// TIA Portal V20 export
DATA_BLOCK "LPFE_GlobalConfigurationData"   // DB240
TITLE = LPFE_GlobalConfigurationData
{ DB_Accessible_From_OPC_UA := 'FALSE' }
AUTHOR : DI FA SUP
FAMILY : LPFE
// Contains all global configurable settings
// stored: Access Published, DBAccessibleFromOPCUA false, DBAccessibleFromWebserver false, MemoryReserve 100, Namespace PFE
   VAR
      globalSessionId { ExternalAccessible := 'False'; ExternalVisible := 'False'; ExternalWritable := 'False'} : UDInt := 123;   // Current session ID echoed in the event messages
      globalPacketIdentifier { ExternalAccessible := 'False'; ExternalVisible := 'False'; ExternalWritable := 'False'} : "LPFE_typeGlobalSeqMgmt";   // ID that is iincremented with each sent message
      globalReceiveDataCounter { ExternalAccessible := 'False'; ExternalVisible := 'False'; ExternalWritable := 'False'; S7_SetPoint := 'True'} : "LPFE_typeGlobalSeqMgmt";   // ID that is incremented with each received message
      globalWriteDataCounter { ExternalAccessible := 'False'; ExternalVisible := 'False'; ExternalWritable := 'False'; S7_SetPoint := 'True'} : "LPFE_typeGlobalSeqMgmt";   // ID that is incremented with each created message
      connectionParametersFromHost { ExternalAccessible := 'False'; ExternalVisible := 'False'; ExternalWritable := 'False'; S7_SetPoint := 'True'} : "LPFE_typeConnectionParameters_1";   // Connection parameters of the FromHost Channel
      connectionParametersToHost { ExternalVisible := 'False'; ExternalWritable := 'False'; S7_SetPoint := 'True'} : Array[0.._.LE_NUMBER_OF_INTERFACE_BUFFERS] of "LPFE_typeConnectionParameters_1";   // Connection parameters of the ToHost Channels
      connectionParametersToHostTxn { ExternalAccessible := 'False'; ExternalVisible := 'False'; ExternalWritable := 'False'; S7_SetPoint := 'True'} : "LPFE_typeConnectionParameters_1";   // Connection parameters of the Txn Channel (Fire-and-Forget)
      channelConfigurationToHost { ExternalVisible := 'False'; S7_SetPoint := 'True'} : Array[0.._.LE_NUMBER_OF_INTERFACE_BUFFERS] of "LPFE_typeRequestChannelConfig";   // toHost Channel Configuration, user can configure the type of messages that can be sent from the channel
      channelConfigurationMQTTToHost : "LPFE_typeRequestChannelConfigMQTT";
      channelConfigurationTxn { ExternalVisible := 'False'; S7_SetPoint := 'True'} : "LPFE_typeOutboundChannelConfig";   // Transaction Channel Configuration
      retryConfiguration { ExternalVisible := 'False'; S7_SetPoint := 'True'} : "LPFE_typeMsgRetryConfig";   // Rettry Configuration Times
      heartbeatConfiguration { ExternalVisible := 'False'} : "LPFE_typeHeartbeatConfig";
      heartbeatInterface : "LPFE_typeHeartbeatInterface";   // Heartbeat signal from Host
      blockingMainBufferDuringResetTime { ExternalAccessible := 'False'; ExternalVisible := 'False'; ExternalWritable := 'False'; S7_SetPoint := 'True'} : Time := T#5s;   // Time in which the buffer will remain blocked after a reset
      cleanupAll { ExternalAccessible := 'False'; ExternalVisible := 'False'; ExternalWritable := 'False'; S7_SetPoint := 'True'} : Bool;   // When set, all message channels are cleared (data loss!) and communication is reset
      shiftInitialization { ExternalWritable := 'False'} : Bool;   // Use this tag to initialize the Shift
      pfeManualReset : Bool;   // Manual Reset for the PFE Mechanism
   END_VAR
BEGIN
   channelConfigurationMQTTToHost.EnableMQTTForTelemetry := TRUE;
   heartbeatConfiguration.incomingHearbeatInterval := t#5s;
   heartbeatConfiguration.outgoingHeartbeatInterval := t#10s;
END_DATA_BLOCK
